(* B8 = Reset *)
TYPE ST_B8Cmd :
STRUCT
	PathID		:UINT	:=0; 		(* 2 bytes*)
	CRC			:UINT   :=0;        (*2 bytes *)     
    //CRC1		:BYTE	:=16#00;    (* 1 byte*)
	//CRC2		:BYTE	:=16#00;    (* 1 byte*)
	
END_STRUCT
END_TYPE

(* stored: Version 1.1.0.1, ProductVersion 3.1.4020.12
   DUT ST_B8Cmd: Id {85e2db18-aa0c-443b-bd3a-e79bfb9c492e} *)
